PROGRAM TableTennisScoreCounter
VAR

	nPlayerOne			:	INT;
	nPlayerTwo			:	INT;
	nPlayerScoreDiff	:	INT;
	
	sPlayerOne			:	STRING;
	sPlayerTwo			:	STRING;
	
	sPlayerList: ARRAY [0..nMaxTableLength] OF STRING := ['Adam', 'Alan', 'Astrid', 'Jamie', 'Ivo', 'Guest'];
		
	sWinner 			: 	STRING;	
	
	xPlayerOneWins		:	BOOL;	
	xPlayerTwoWins		:	BOOL;	
	
	rtPlayerOne			:	R_TRIG;	
	rtPlayerTwo			:	R_TRIG;
	rtResetOne			:	R_TRIG;
	rtResetTwo			:	R_TRIG;
	
	gameMode5s			:	BOOL;
	
	i: INT;
END_VAR

rtPlayerOne(CLK := PTM200StrippedTables[12].Signal);
rtPlayerTwo(CLK := PTM200StrippedTables[13].Signal);
rtResetOne(CLK := PTM200StrippedTables[14].Signal);
rtResetTwo(CLK := PTM200StrippedTables[15].Signal);



IF rtPlayerOne.Q THEN
	nPlayerOne := nPlayerOne + 1;
END_IF

IF rtPlayerTwo.Q THEN
	nPlayerTwo := nPlayerTwo + 1;
END_IF

IF rtResetOne.Q THEN
	nPlayerOne := 0;
END_IF

IF rtResetTwo.Q THEN
	nPlayerTwo := 0;
END_IF

IF gameMode5s THEN
	Play5s();
ELSE
	Play11s();
END_IF

nPlayerScoreDiff := ABS(nPlayerOne - nPlayerTwo);

IF nPlayerOne >= 11 AND nPlayerOne > nPlayerTwo AND nPlayerScoreDiff >= 2 THEN
	sWinner := CONCAT(sPlayerOne, ' Wins');
	xPlayerOneWins := TRUE;
ELSIF nPlayerTwo >= 11 AND nPlayerTwo > nPlayerOne AND nPlayerScoreDiff >= 2 THEN
	sWinner := CONCAT(sPlayerTwo, ' Wins');
	xPlayerTwoWins := TRUE;
END_IF

IF nPlayerOne = 0 AND  nPlayerTwo = 0 THEN
	sWinner := '';
	xPlayerOneWins := FALSE;
	xPlayerTwoWins := FALSE;
END_IF

FOR i := 5 TO 49 DO //Set to 5 so as not to overwrite staff names

	IF 	CurrentMonthSignInTable[i].Name = '' THEN
	sPlayerList[i] := CurrentMonthSignInTable[i-5].Name;
	ELSE
	EXIT;	
	END_IF

END_FOR

ACTION Play11s:

END_ACTION

ACTION Play5s:

END_ACTION

END_PROGRAM

(* stored: Version 1.1.0.1, ProductVersion 3.1.4024.12
   POU TableTennisScoreCounter: Id {6768a184-5b20-4146-a9d5-4c417992d68d}, SpecialFunc None
   Action Play11s: Id {dc62f77a-2645-45c3-84aa-a9111567b17c}
   Action Play5s: Id {3f4e4df5-95f4-4973-8294-4fd554bd3829} *)
